FUNCTION_BLOCK FB_ModbusMaster_Test EXTENDS FB_TestSuite

VAR
END_VAR

END_FUNCTION_BLOCK

(* stored: Version 1.1.0.1, ProductVersion 3.1.4024.12
   POU FB_ModbusMaster_Test: Id {b7e169e6-23e0-47cc-bba5-b3ea5eb58bcc}, SpecialFunc None *)
